// TIA Portal project "llenado_automatico" (V18)
// Proceso de llenado automatico simple

(* hardware
DEVICE "S7-1200 station_1"  S7-1200 Station
   slot 0: "Rack_0"  S7-1200 Rack  Rack  V1.0
   slot 1: "PLC_1"  CPU 1212C AC/DC/Rly  6ES7 212-1BE40-0XB0  V4.6
*)

// ===== PLC "PLC_1"  CPU 1212C AC/DC/Rly =====

VAR_GLOBAL   // PLC tag table "In/Out"
   "In" AT %I0.0 : "Inputs";
   "Out" AT %Q0.0 : "Outputs";
END_VAR

TYPE "Inputs"
   STRUCT
      PB_Start : Bool;   // Pushbutton Start normally open
      PB_stop : Bool;   // Pushbutton Stop normally close
      Level_box_sensor : Bool;   // Hihg level sensor box normally open
      Position_sensor : Bool;   // Position box sensor normally open
      Low_level_hopper : Bool;   // Low leven hopper sensor normally open
   END_STRUCT;
END_TYPE

TYPE "Outputs"
   STRUCT
      Conveyor : Bool;   // Motor conveyor
      Run_pilot : Bool;   // Run indicator pilot
      Standby_pilot : Bool;   // Standby indicator pilot
      Full_pilot : Bool;   // Full indicator pilot
      Solenoid : Bool;   // Solenoid valve
   END_STRUCT;
END_TYPE

DATA_BLOCK "Global_var"   // DB1
{ S7_Optimized_Access := 'TRUE' }
AUTHOR : Stiven Perez Mora
VERSION : 0.1
   VAR
      In : "Inputs";
      Out : "Outputs";
      Start_Stop_Process : Bool;
   END_VAR
BEGIN
END_DATA_BLOCK

FUNCTION "Start_Stop_Process" : Void   // FC1, LAD
TITLE = Start Stop process
{ S7_Optimized_Access := 'TRUE' }
AUTHOR : Stiven Perez Mora
VERSION : 0.1
// Condition to start stop process
   VAR_INPUT
      Start : Bool;
      Stop : Bool;
      Level_Sensor_Hopper : Bool;
   END_VAR
   VAR_IN_OUT
      Standby_pilot : Bool;   // Standby pilot indicator
      Run_pilot : Bool;   // Run pilot indicator
   END_VAR
BEGIN

REGION Network 1: Start Process
   // condition to start process and activate run pilot indicator
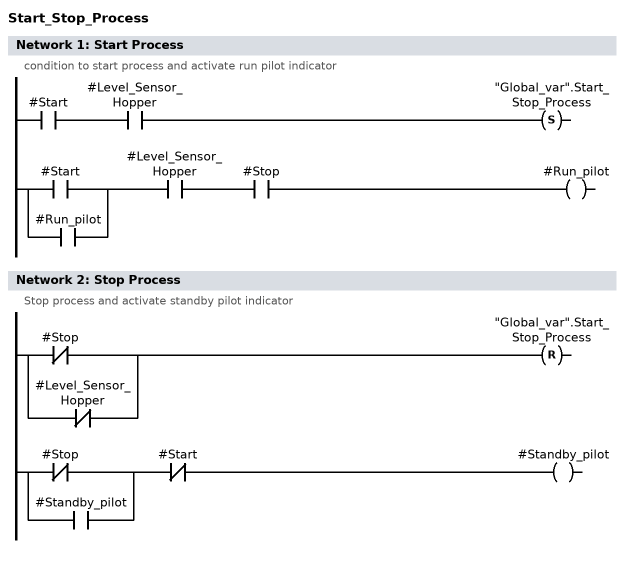
   RUNG wire#powerrail
      Contact( #Start )
      Contact( #Level_Sensor_Hopper )
      S_Coil( "Global_var".Start_Stop_Process )
   END_RUNG
   RUNG wire#powerrail
      Contact( #Start )
      wire#w1
      Contact( #Level_Sensor_Hopper )
      Contact( #Stop )
      Coil( #Run_pilot )
   END_RUNG
   RUNG wire#powerrail
      Contact( #Run_pilot )
   END_RUNG wire#w1
   // the same network as SCL:
   IF #Start AND #Level_Sensor_Hopper THEN "Global_var".Start_Stop_Process := TRUE; END_IF;
   #Run_pilot := (#Start OR #Run_pilot) AND #Level_Sensor_Hopper AND #Stop;
END_REGION

REGION Network 2: Stop Process
   // Stop process and activate standby pilot indicator
   RUNG wire#powerrail
      I_Contact( #Stop )
      wire#w1
      R_Coil( "Global_var".Start_Stop_Process )
   END_RUNG
   RUNG wire#powerrail
      I_Contact( #Level_Sensor_Hopper )
   END_RUNG wire#w1
   RUNG wire#powerrail
      I_Contact( #Stop )
      wire#w2
      I_Contact( #Start )
      Coil( #Standby_pilot )
   END_RUNG
   RUNG wire#powerrail
      Contact( #Standby_pilot )
   END_RUNG wire#w2
   // the same network as SCL:
   IF NOT #Stop OR NOT #Level_Sensor_Hopper THEN "Global_var".Start_Stop_Process := FALSE; END_IF;
   #Standby_pilot := (NOT #Stop OR #Standby_pilot) AND NOT #Start;
END_REGION
END_FUNCTION

FUNCTION "Fill_Process" : Void   // FC2, LAD
TITLE = Fill Process
{ S7_Optimized_Access := 'TRUE' }
AUTHOR : Stiven Perez Mora
VERSION : 0.1
// Condition to fill process
   VAR_INPUT
      Position_sensor : Bool;   // Position box sensor normally open
      Level_box_sensor : Bool;   // High level box sensor normally open
   END_VAR
   VAR_OUTPUT
      Conveyor : Bool;   // Motor conveyor
      Solenoid : Bool;   // solenoid hopper
      Full_pilot : Bool;   // Full pilot indicator, high level box
   END_VAR
BEGIN

REGION Network 1: Activate Motor conveyor
   // Conditions to activate and deactive motor conveyor
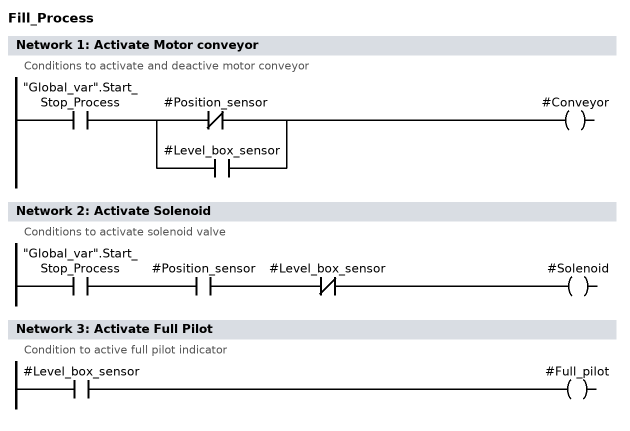
   RUNG wire#powerrail
      Contact( "Global_var".Start_Stop_Process )
      wire#w1
      I_Contact( #Position_sensor )
      wire#w2
      Coil( #Conveyor )
   END_RUNG
   RUNG wire#w1
      Contact( #Level_box_sensor )
   END_RUNG wire#w2
   // the same network as SCL:
   #Conveyor := "Global_var".Start_Stop_Process AND (NOT #Position_sensor OR #Level_box_sensor);
END_REGION

REGION Network 2: Activate Solenoid
   // Conditions to activate solenoid valve
   RUNG wire#powerrail
      Contact( "Global_var".Start_Stop_Process )
      Contact( #Position_sensor )
      I_Contact( #Level_box_sensor )
      Coil( #Solenoid )
   END_RUNG
   // the same network as SCL:
   #Solenoid := "Global_var".Start_Stop_Process AND #Position_sensor AND NOT #Level_box_sensor;
END_REGION

REGION Network 3: Activate Full Pilot
   // Condition to active full pilot indicator
   RUNG wire#powerrail
      Contact( #Level_box_sensor )
      Coil( #Full_pilot )
   END_RUNG
   // the same network as SCL:
   #Full_pilot := #Level_box_sensor;
END_REGION
END_FUNCTION

ORGANIZATION_BLOCK "Main"   // OB1, LAD, ProgramCycle
TITLE = "Main Program Sweep (Cycle)"
{ S7_Optimized_Access := 'TRUE' }
VERSION : 0.1
   VAR_INPUT
      Initial_Call : Bool;   // Initial call of this OB
      Remanence : Bool;   // =True, if remanent data are available
   END_VAR
BEGIN

REGION Network 1: Start stop process block
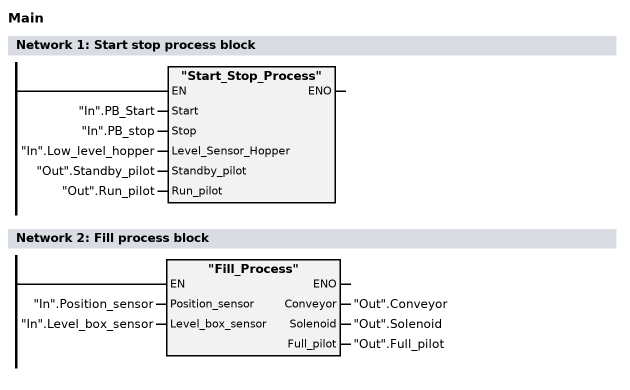
   RUNG wire#powerrail
      "Start_Stop_Process"(Start := "In".PB_Start, Stop := "In".PB_stop, Level_Sensor_Hopper := "In".Low_level_hopper, Standby_pilot := "Out".Standby_pilot, Run_pilot := "Out".Run_pilot)
   END_RUNG
   // the same network as SCL:
   "Start_Stop_Process"(Start := "In".PB_Start,
                        Stop := "In".PB_stop,
                        Level_Sensor_Hopper := "In".Low_level_hopper,
                        Standby_pilot := "Out".Standby_pilot,
                        Run_pilot := "Out".Run_pilot);
END_REGION

REGION Network 2: Fill process block
   RUNG wire#powerrail
      "Fill_Process"(Position_sensor := "In".Position_sensor, Level_box_sensor := "In".Level_box_sensor, Conveyor => "Out".Conveyor, Solenoid => "Out".Solenoid, Full_pilot => "Out".Full_pilot)
   END_RUNG
   // the same network as SCL:
   "Fill_Process"(Position_sensor := "In".Position_sensor,
                  Level_box_sensor := "In".Level_box_sensor,
                  Conveyor => "Out".Conveyor,
                  Solenoid => "Out".Solenoid,
                  Full_pilot => "Out".Full_pilot);
END_REGION
END_ORGANIZATION_BLOCK